Fanuc KAREL source: compact_preamble.KL

PROGRAM KB00195
%NOLOCKGROUP
VAR
P1 : STRING[80];P2 : STRING[80];P3:INTEGER;P4:INTEGER;P5:INTEGER;P6 : ARRAY[4] OF STRING[80];P7:INTEGER;P8:INTEGER
BEGIN
P1='A'
P2='A'
P3=1
P4=1
P5=1
P7=1
P8=1
VAR_LIST(P1,P2,P3,P4,P5,P6,P7,P8)
END KB00195
